// Mitsubishi GX Works2 project: wandEx01   PLC: Q02/Q02H

PROGRAM MAIN
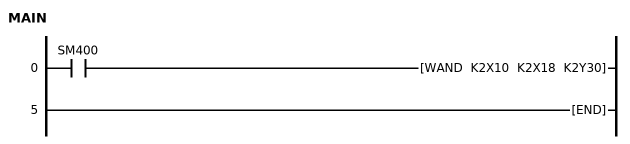
0     LD      SM400
      WAND    K2X10 K2X18 K2Y30
5     END
END_PROGRAM
